# B&R Automation Studio project RSD
Automation Studio 4.3.3.196

## Configuration RSD_Default

CPU X20CP1382, AutomationRuntime I4.33, Build 4.1.2, Vc V4.33.0

### Task classes (Cpu.sw)
```
Cyclic#1 (cycle 2000 us, tolerance 2000 us):
  RSI <- RSI.prg
  Camera <- Camera.prg
Cyclic#2 (cycle 10000 us, tolerance 10000 us):
  Servo <- Servo.prg
  MES_Comm <- MES_Comm.prg
Cyclic#3 (cycle 20000 us, tolerance 20000 us):
  Camera_A <- Camera_A.prg
Cyclic#4:
  Feeder <- Feeder.prg
  Conveyor <- Conveyor.prg
Binaries: udbdef, TCData, ashwac, arconfig, asfw, ashwd, iomap, User, Role, sysconf
Libraries: AsHttp, runtime, AsTCP, AsUDP, standard, MTBasics, brsystem, MTTypes, sys_lib, astime, asieccon
```

### Hardware
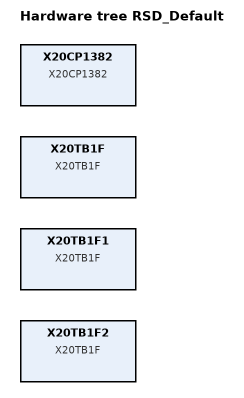
```
X20CP1382 : X20CP1382 v1.3.2.0  [X1 -> X1.SL; X2 -> X2.SL; X3 -> X3.SL]
  Module X1 (Type=X1, Virtual=true, Version=1.3.2.0)
    Connection (Connector=SS1, TargetModule=X20TB1F, TargetConnector=SS)
    Connection (Connector=SL, TargetModule=X20CP1382, TargetConnector=X1)
  Module X2 (Type=X2, Virtual=true, Version=1.3.2.0)
    Connection (Connector=SS1, TargetModule=X20TB1F1, TargetConnector=SS)
    Connection (Connector=SL, TargetModule=X20CP1382, TargetConnector=X2)
  Module X3 (Type=X3, Virtual=true, Version=1.3.2.0)
    Connection (Connector=SS1, TargetModule=X20TB1F2, TargetConnector=SS)
    Connection (Connector=SL, TargetModule=X20CP1382, TargetConnector=X3)
    X3Channel09Source = PWMout
  Connector IF2:
    ActivateDevice = 1
    Mode = Manual
    InternetAddress = 192.168.1.80
    SubnetMask = 255.255.255.0
    InaNodeNumber = 0
  ConfigurationID = RSD_RSD_Default
  SystemTick = 1000
  TaskClassIdleTime = 5000
  CyclicTaskClassCount = 4
  Cyclic1Duration = 2000
  Cyclic1Tolerance = 2000
  Cyclic1Stack = 16384
  Cyclic2Duration = 10000
  Cyclic2Tolerance = 10000
  Cyclic3Duration = 20000
  Cyclic3Tolerance = 20000
X20TB1F : X20TB1F v1.0.0.0
X20TB1F1 : X20TB1F v1.0.0.0
X20TB1F2 : X20TB1F v1.0.0.0
```

### IoMap.iom - X20CP1382/IoMap.iom
```iecst
VAR_CONFIG
	::Camera_A:Camera_trigger AT %QX."X3".DigitalOutput01;
	::Conveyor:Conveyor_out AT %QX."X3".DigitalOutput02;
	::Enable_in AT %IX."X2".DigitalInput01;
	::Sensor_in AT %IX."X2".DigitalInput02;
	::Servo:Period AT %QW."X3".PWMPeriod09;
	::Servo:Pulse AT %QW."X3".PWMOutput09;
	::Feeder:Output_signal AT %QX."X3".DigitalOutput03;
	::Feeder:Enable_feeder AT %IX."X2".DigitalInput09;
END_VAR
```

## Logical view

Binary libraries used (declarations not repeated): operator, runtime, astime, AsIecCon, AsHttp, AsTCP, AsUDP, standard, MTBasics 2.21.0, brsystem, MTTypes 1.03.4, sys_lib, asstring

### Global.var - Global variables
```iecst
VAR
	Camera_bad : BOOL := FALSE;
	Enable_in : BOOL;
	Sensor_in : BOOL;
	Camera_good : BOOL := FALSE;
	Tilt : BOOL := FALSE;
	Data_send : STRING[200] := '';
	Data_recv_vector : ARRAY[0..9] OF STRING[4];
	data_received : BOOL := FALSE;
	New_data : BOOL := FALSE;
	Data_recv_index : USINT := 0;
	Current_part_id : UDINT;
	Part_selected : BOOL := FALSE;
	Data_length : USINT;
	Should_recv : BOOL := FALSE;
	Current_part_post : BOOL := FALSE;
	Robot_index : STRING[2];
	Ready : STRING[1];
	Activate_override : BOOL := TRUE;
	Buffer_use : STRING[1] := '0';
	Activate : BOOL := FALSE;
END_VAR
```

### Global2.typ
```iecst
TYPE
	Variables : 	STRUCT
		isGoodCounter : USINT;
		isBadCounter : USINT;
		position : UDINT;
		sliske : UDINT;
		buffer_bad : ARRAY[0..4]OF UDINT;
		buffer_good : ARRAY[0..10]OF UDINT;
	END_STRUCT;
END_TYPE
```


### Program Logical/Camera_A (IEC)

#### Variables.var
```iecst
VAR
	Delay : MTBasicsTimeDelay;
	Camera_trigger : BOOL := TRUE;
END_VAR
```

#### Main.st
```iecst
PROGRAM _INIT
	(* Insert code here *)
	Delay.Enable := TRUE;
	Delay.DelayTime := 0.227; // 1 at 10hz, 0.4 at 20hz

END_PROGRAM

PROGRAM _CYCLIC
	(* Insert code here *)

	IF Enable_in = TRUE THEN
		Delay.In := BOOL_TO_REAL(Sensor_in);
		Delay();
		Camera_trigger := REAL_TO_BOOL(Delay.Out);
	ELSE
		Camera_trigger := FALSE;
	END_IF

END_PROGRAM

PROGRAM _EXIT
	(* Insert code here *)

END_PROGRAM
```

### Program Logical/Conveyor (IEC)

#### Variables.var
```iecst
VAR
	Conveyor_out : BOOL := FALSE;
END_VAR
```

#### Cyclic.st
```iecst
PROGRAM _CYCLIC
	(* Insert code here *)
	Conveyor_out := Enable_in;

END_PROGRAM
```

#### Init.st
```iecst
PROGRAM _INIT
	(* Insert code here *)

END_PROGRAM
```

### Program Logical/MES_Comm (IEC)

#### Client.st - Cyclic code
```iecst
(********************************************************************
 * COPYRIGHT -- Bernecker + Rainer
 ********************************************************************
 * Program: Client
 * File: Client.st
 * Author: Bernecker + Rainer
 * Created: February 21, 2008
 ********************************************************************
 * Implementation of program Client
 ********************************************************************)
PROGRAM _INIT

END_PROGRAM
PROGRAM _CYCLIC

	CASE Client.sStep OF

		 3: (* IDLE state - waits here until there is something to send *)
			IF New_data <> FALSE THEN
				Client.sStep:=20;
			END_IF;

		 0: (* Open Ethernet Interface *)
			Client.TcpOpen_0.enable := 1;
			Client.TcpOpen_0.pIfAddr := 0;  (* Which Interface to open *)
			Client.TcpOpen_0.port := 13001;  (* Port on client side to use *)
			Client.TcpOpen_0.options :=  0;
			Client.TcpOpen_0;  (* Call the Function *)

			IF Client.TcpOpen_0.status = 0 THEN  (* TcpOpen successfull *)
				Client.sStep := 5;
			ELSIF Client.TcpOpen_0.status = ERR_FUB_BUSY THEN  (* TcpOpen not finished -> redo *)
			  (* Busy *)
			ELSE  (* Goto Error Step *)
				Client.sStep := 100;
			END_IF

		 5:
		 	Client.linger_opt.lLinger := 0; (* linger Time = 0 *)
			Client.linger_opt.lOnOff := 1; (* linger Option ON *)

		 	Client.TcpIoctl_0.enable := 1;
			Client.TcpIoctl_0.ident := Client.TcpOpen_0.ident; (* Connection Ident from AsTP.TCP_Open *)
			Client.TcpIoctl_0.ioctl := tcpSO_LINGER_SET; (* Set Linger Options *)
			Client.TcpIoctl_0.pData := ADR(Client.linger_opt);
			Client.TcpIoctl_0.datalen := SIZEOF(Client.linger_opt);
   			Client.TcpIoctl_0;

			IF Client.TcpIoctl_0.status = 0 THEN  (* TcpIoctl successfull *)
				Client.sStep := 10;
			ELSIF Client.TcpIoctl_0.status = ERR_FUB_BUSY THEN  (* TcpIoctl not finished -> redo *)
			  (* Busy *)
			ELSE  (* Goto Error Step *)
				Client.sStep := 100;
			END_IF

		10: (* Connect to the other Station *)
			Client.TcpClient_0.enable := 1;
			Client.TcpClient_0.ident := Client.TcpOpen_0.ident;  (* Connection Ident from AsTCP.TCP_Open *)
			Client.TcpClient_0.portserv := 4567;  (* Port on server side to use *)
			Client.TcpClient_0.pServer := ADR('192.168.1.23');  (* Server Address *)
			Client.TcpClient_0;  (* Call the Function*)

			IF Client.TcpClient_0.status = 0 THEN  (* Open ok -> Send Data *)
				Client.sStep := 3;
			ELSIF Client.TcpClient_0.status = ERR_FUB_BUSY THEN  (* TcpClient not finished -> redo *)
			  (* Busy *)
			ELSIF Client.TcpClient_0.status = tcpERR_INVALID THEN  (* Port error -> Close actual connection, and reopen a new one *)
				Client.sStep := 40;
			ELSE  (* Goto Error Step *)
				Client.sStep := 100;
			END_IF

		20: (* Send Data to the Server *)
			Client.TcpSend_0.enable := 1;
			Client.TcpSend_0.ident := Client.TcpOpen_0.ident;  (* Connection Ident from AsTCP.TCP_Open *)
			Client.TcpSend_0.pData := ADR(Data_send);  (* Which data to send *)
			Client.TcpSend_0.datalen := Data_length; //SIZEOF(Data_send);  (* Lenght of data to send *)
			Client.TcpSend_0.flags := 0;
			Client.TcpSend_0;  (* Call the Function*)
			Data_recv_index := 0;
			FOR counter:=0 TO 9 BY 1 DO
				Data_recv_vector[counter] := '';
			END_FOR

			IF Client.TcpSend_0.status = 0 THEN  (* Data was sent sucessfully -> receive data *)
				New_data:=FALSE;
				IF Should_recv THEN
					Client.sStep := 30;
				ELSE
					Client.sStep := 3;
				END_IF

			ELSIF Client.TcpSend_0.status = ERR_FUB_BUSY THEN  (* TcpSend not finished -> redo *)
			  (* Busy *)
			ELSIF (Client.TcpSend_0.status = tcpERR_SENTLEN) OR (Client.TcpSend_0.status = tcpERR_NOT_CONNECTED) THEN (* Connection Lost *)
				Client.sStep := 40;
			ELSE  (* Goto Error Step *)
				Client.sStep := 100;
			END_IF

	    30: (* Receive Data from the Server *)
			Client.TcpRecv_0.enable := 1;
			Client.TcpRecv_0.ident := Client.TcpOpen_0.ident;  (* Connection Ident from AsTCP.TCP_Open *)
			Client.TcpRecv_0.pData	:= ADR(Data_recv_vector[Data_recv_index]);  (* Where to store the incoming data *)
			Client.TcpRecv_0.datamax := SIZEOF(Data_recv_vector[Data_recv_index]);  (* Lenght of data buffer *)
			Client.TcpRecv_0.flags := 0;
			Client.TcpRecv_0;  (* Call the Function*)

			IF Client.TcpRecv_0.status = 0 THEN  (* Data was received sucessfully -> Send next packet *)
				Client.sStep := 30;
				Client.recv_timeout := 0;

				//Data_recv_vector[Data_recv_index] := Data_recv;
				Data_recv_index := Data_recv_index +1;
			ELSIF Client.TcpRecv_0.status = tcpERR_NO_DATA THEN  (* No data received - wait *)
				Client.recv_timeout := Client.recv_timeout + 1;
				IF Client.recv_timeout > 10 THEN
					Client.sStep := 3;
					Client.recv_timeout := 0;
					data_received := TRUE;
				END_IF

				(* No Data received *)
			ELSIF Client.TcpRecv_0.status = ERR_FUB_BUSY THEN  (* TcpRecv not finished -> redo *)
				(* Busy *)
			ELSIF Client.TcpRecv_0.status = tcpERR_NOT_CONNECTED THEN (* Connection Lost *)
				Client.sStep := 40;
			ELSE  (* Goto Error Step *)
				Client.sStep := 100;
			END_IF

		40: (* Close connection *)
			Client.TcpClose_0.enable := 1;
			Client.TcpClose_0.ident := Client.TcpOpen_0.ident;  (* Connection Ident from AsTCP.TCP_Open *)
			Client.TcpClose_0.how := 0;
			Client.TcpClose_0;  (* Call the Function*)

			IF Client.TcpClose_0.status = 0 THEN  (* Close sucessfull -> Reopen the interface *)
				Client.sStep := 3;
			ELSIF Client.TcpClose_0.status = ERR_FUB_BUSY THEN  (* TcpClose not finished -> redo *)
			  (* Busy *)
			ELSE  (* Goto Error Step *)
				Client.sStep := 100;
			END_IF

	   100: (* Here some error Handling has to be implemented *)

	END_CASE

END_PROGRAM
```

#### Client.var - Data for Client Task
```iecst
(********************************************************************
 * COPYRIGHT -- Bernecker + Rainer
 ********************************************************************
 * Package: LibAsTCP
 * File: LibAsTCP.var
 * Author: Bernecker + Rainer
 * Created: February 21, 2008
 ********************************************************************
 * Variables of package LibAsTCP
 ********************************************************************)
VAR
	Client : Client_typ := (0); (*Data for Client Task*)
	State_send : USINT := 0;
	counter : USINT;
END_VAR
```

#### Variables.var - not listed in the package file held
```iecst
VAR
	Client : httpClient;
	Enable : BOOL := TRUE;
	Send : BOOL := FALSE;
	IP : STRING[80] := '192.168.1.23';
	URI : STRING[80] := '/plc.test';
	RESPONSE : STRING[4096];
	REQUESTLENGTH : UDINT := 0;
	REQUESTDATA : STRING[80];
	RESPONSELENGTH : UDINT := 4096;
END_VAR
```

#### Cyclic.st - not listed in the package file held
```iecst
PROGRAM _CYCLIC
	(* Insert code here *)
	Client.enable := Enable;

	Client.send := Send;

	Client();

END_PROGRAM
```

#### Init.st - not listed in the package file held
```iecst
PROGRAM _INIT
	(* Insert code here *)
	Client.hostPort := 80;
	Client.method := httpMETHOD_GET;
	Client.option := httpOPTION_HTTP_11;
	Client.pHost := ADR(IP);
	Client.pUri := ADR(URI);
	Client.pRequestData := ADR(REQUESTDATA);
	Client.requestDataLen := REQUESTLENGTH;
	Client.pResponseData := ADR(RESPONSE);
	Client.responseDataSize := RESPONSELENGTH;

END_PROGRAM
```

### Program Logical/MES_machine (IEC)

#### Main.st - Init, cyclic, exit code
```iecst
PROGRAM _INIT
	(* Insert code here *)

END_PROGRAM

PROGRAM _CYCLIC
	(* Insert code here *)

	CASE MES_step OF

		0:		// ST-Start
			Part_selected := FALSE;
			data_received := FALSE;

		5:		// ST-Idle
			IF Order_selected = FALSE THEN
				MES_step := 20;

			ELSIF Part_selected = FALSE AND Sensor_in THEN
				MES_step := 10;

			ELSIF Current_part_post = FALSE AND (Camera_good OR Camera_bad) THEN
				MES_step := 15;

			ELSIF Part_status_posted THEN
				IF Camera_good AND Order_good > 0 THEN
					MES_step := 30;
				ELSIF Camera_bad AND Order_bad > 0 THEN
					MES_step := 30;
				ELSIF Camera_good AND buffer_free(ADR(variables), TRUE) THEN
					MES_step := 40;
				ELSIF Camera_bad AND buffer_free(ADR(variables), FALSE) THEN
					MES_step := 40;
				ELSE
					MES_step := 43;

				END_IF

				Part_status_posted := FALSE;
			END_IF

		10:		// ST-Get part
			IF New_data = FALSE THEN
				Data_send := 'GET PART 1$n';
				Data_length := 11;
				New_data := TRUE;
				MES_step := 11;
				Should_recv := TRUE;
				Activate_override := TRUE;
			END_IF

		11:
			IF data_received = TRUE THEN
				data_received := FALSE;
				memcpy(ADR(Current_part_id), ADR(Data_recv_vector[0]),4);
				Part_selected := TRUE;
				Current_part_post := FALSE;
				MES_step := 5;
			END_IF

		15:		// ST-Post Part
			IF New_data = FALSE THEN
				Data_send := 'POST PARTSTATUS$n';
				Number := 1000;
				WHILE Number > Current_part_id AND Number <> 0 DO
					Data_send:=CONCAT(Data_send, '0');
					Number := Number/10;
				END_WHILE;

				IF Current_part_id <> 0 THEN
					String_tmp := UDINT_TO_STRING(Current_part_id);
					Data_send:=CONCAT(Data_send, String_tmp);
				END_IF

				IF Camera_good THEN
					Data_send:=CONCAT(Data_send, ' 1$n');
				ELSIF Camera_bad THEN
					Data_send:=CONCAT(Data_send, ' 0$n');
				END_IF

				Data_length := 23;
				Should_recv := FALSE;
				New_data := TRUE;
				Part_selected := FALSE;
				Current_part_post := TRUE;
				MES_step := 5;
				Part_status_posted := TRUE;
			END_IF

		20:		// ST-Get Order
			IF New_data = FALSE THEN
				Data_send := 'GET ORDER 1$n';
				Data_length := 12;
				Current_order_ids := '';
				New_data := TRUE;
				MES_step := 21;
				Should_recv := TRUE;
			END_IF

		21:
			IF data_received = TRUE THEN
				data_received := FALSE;
				memcpy(ADR(Current_order_id), ADR(Data_recv_vector[0]),4);
				IF Current_order_id > 10000 THEN
					MES_step := 45;
				ELSE
					Order_good := 0;
					Order_bad := 0;
					memcpy(ADR(Current_order_parts), ADR(Data_recv_vector[1]),4);
					FOR Order_index:=0 TO Current_order_parts-1 BY 1 DO
						memcpy(ADR(Parts_vector[Order_index]), ADR(Data_recv_vector[Order_index+2]),4);
						IF Parts_vector[Order_index] = 1 THEN
							Order_good := Order_good +1;
						ELSIF Parts_vector[Order_index] = 0 THEN
							Order_bad := Order_bad +1;
						END_IF

					END_FOR

					Order_selected := TRUE;
						MES_step := 5;

				END_IF

			END_IF

		25:		// ST-Post Order
			IF New_data = FALSE THEN
				Data_send := 'POST ORDERSTATUS$n';
				Number := 1000;
				WHILE Number > Current_order_id AND Number <> 0 DO
					Data_send:=CONCAT(Data_send, '0');
					Number := Number/10;
				END_WHILE;

				IF Current_order_id <> 0 THEN
					String_tmp := UDINT_TO_STRING(Current_order_id);
					Data_send:=CONCAT(Data_send, String_tmp);
				END_IF

				Data_length := 21;
				Data_send := CONCAT(Data_send, Current_order_ids);
				Current_order_ids := CONCAT(Current_order_ids, 'p');
				Pos_find := FIND(Current_order_ids, 'p');
				Data_length := Data_length + INT_TO_USINT(Pos_find);

				Data_send := CONCAT(Data_send, '$n');
				Should_recv := FALSE;
				New_data := TRUE;
				Order_selected := FALSE;
				MES_step := 5;
			END_IF

		30:		// ST - Put box
			Buffer_use := '0';
			Robot_index := '0';
			String_tmp := UDINT_TO_STRING(Current_part_id);
			Current_order_ids := CONCAT(Current_order_ids, String_tmp);
			Current_order_ids := CONCAT(Current_order_ids, ' ');
			IF Camera_good THEN
				Order_good := Order_good - 1;
			ELSIF Camera_bad THEN
				Order_bad := Order_bad -1;
			END_IF;
			MES_step := 31;

		31:
			IF Ready = '0' THEN
				MES_step := 32;
			END_IF;

		32:
			IF Ready = '1' THEN
				IF Order_good = 0 AND Order_bad = 0 THEN
					Tilt := TRUE;
					MES_step := 25;
				ELSIF Order_good > 0 AND in_buffer(ADR(variables),TRUE) THEN
					MES_step := 35;
				ELSIF Order_bad > 0 AND in_buffer(ADR(variables), FALSE) THEN
					MES_step := 35;
				ELSE
					MES_step := 5;
				END_IF

			END_IF;

		35:		// ST- Tak Buf
			Buffer_use := '0';
			IF Order_good > 0 AND in_buffer(ADR(variables), TRUE) THEN
				Robot_index := UDINT_TO_STRING(fetch_brick_decimal(ADR(variables), TRUE));
				Buffer_part_id := get_partid(ADR(variables), TRUE, variables.isGoodCounter);
				Order_good := Order_good - 1;
			ELSIF Order_bad > 0 AND in_buffer(ADR(variables), FALSE) THEN
				Robot_index := UDINT_TO_STRING(fetch_brick_decimal(ADR(variables), FALSE));
				Buffer_part_id := get_partid(ADR(variables), FALSE, variables.isBadCounter);
				Order_bad := Order_bad - 1;
			END_IF

			Activate := TRUE;

			String_tmp := UDINT_TO_STRING(Buffer_part_id);
			Current_order_ids := CONCAT(Current_order_ids, String_tmp);
			Current_order_ids := CONCAT(Current_order_ids, ' ');
			MES_step := 36;

		36:
			IF Ready = '0' THEN
				MES_step := 37;
			END_IF

		37:
			IF Ready = '1' THEN
				IF Order_good = 0 AND Order_bad = 0 THEN
					Tilt := TRUE;
					MES_step := 25;
				ELSE
					MES_step := 5;
				END_IF
			END_IF

		40:		// ST- put buf

			IF Camera_good AND buffer_free(ADR(variables), TRUE) THEN
				Buffer_use := '1';
				Robot_index := UDINT_TO_STRING(save_brick_decimal(ADR(variables), TRUE, Current_part_id));
			ELSIF Camera_bad AND buffer_free(ADR(variables), FALSE) THEN
				Buffer_use := '1';
				Robot_index := UDINT_TO_STRING(save_brick_decimal(ADR(variables), FALSE, Current_part_id));
			END_IF
			MES_step := 41;

		41:
			IF Ready = '0' THEN
				MES_step := 42;
			END_IF;

		42:
			IF Ready = '1' THEN
				MES_step := 5;
			END_IF

		43: // BUF full
			Activate_override := FALSE;

			IF New_data = FALSE THEN
				Data_send := 'POST PARTSTATUS$n';
				Number := 1000;
				WHILE Number > Current_part_id AND Number <> 0 DO
					Data_send:=CONCAT(Data_send, '0');
					Number := Number/10;
				END_WHILE;

				IF Current_part_id <> 0 THEN
					String_tmp := UDINT_TO_STRING(Current_part_id);
					Data_send:=CONCAT(Data_send, String_tmp);
				END_IF

				Data_send:= CONCAT(Data_send, ' Buffer full$n');

				Data_length := 33;
				Should_recv := FALSE;
				New_data := TRUE;
				MES_step := 5;
			END_IF

		45:		// ST- Finished
			Activate_override := FALSE;

	END_CASE

END_PROGRAM

PROGRAM _EXIT
	(* Insert code here *)

END_PROGRAM
```

#### Variables2.var - Local variables
```iecst
VAR
	MES_step : USINT := 0;
	Number : UDINT;
	Pos_find : INT;
	String_tmp : STRING[200];
	Current_order_id : UDINT;
	Order_selected : BOOL := FALSE;
	Current_order_parts : UDINT;
	Order_index : UDINT;
	Parts_vector : ARRAY[0..4] OF UDINT;
	Order_good : UDINT;
	Order_bad : UDINT;
	Part_status_posted : BOOL := FALSE;
	Current_order_ids : STRING[200];
	Part_moved : BOOL := FALSE;
	Buffer_part_id : UDINT;
END_VAR
```

#### buffer_free.st
```iecst
(* TODO: Add your comment here *)
FUNCTION buffer_free
	IF type THEN
		IF var.isGoodCounter < 10 THEN
			buffer_free:= TRUE;
		ELSE
			buffer_free:=FALSE;
		END_IF;
	END_IF;

	IF type = FALSE THEN
		IF var.isBadCounter < 5 THEN
			buffer_free:= TRUE;
		ELSE
			buffer_free:=FALSE;
		END_IF;
	END_IF;
END_FUNCTION
```

#### fetch_brick.st
```iecst
FUNCTION fetch_brick
	IF type THEN
		IF var.isGoodCounter <> 0 THEN
			fetch_brick:=var.isGoodCounter;
			var.isGoodCounter:=var.isGoodCounter-1;
		ELSE
			fetch_brick:=-1; // Empty
		END_IF;
	ELSE
		IF var.isBadCounter <> 0 THEN
			fetch_brick:=var.isBadCounter;
			var.isBadCounter:=var.isBadCounter-1;
		ELSE
			fetch_brick:=-1; // Empty
		END_IF;
	END_IF;
END_FUNCTION
```

#### fetch_brick_decimal.st
```iecst
(* TODO: Add your comment here *)
FUNCTION fetch_brick_decimal
	var.position := fetch_brick(ADR(var), type);

	IF var.position = -1 THEN
		fetch_brick_decimal := -1;
		RETURN;
	END_IF;

	IF type = FALSE THEN
		var.sliske:=2;
	ELSE
		IF var.position > 5 THEN
			var.sliske:=3;
		ELSE
			var.sliske:=1;
		END_IF;
	END_IF;

	IF var.position > 5 THEN
		fetch_brick_decimal := SHL(var.sliske,3) + var.position -5 -1;
	ELSE
		fetch_brick_decimal := SHL(var.sliske,3) + var.position -1;
	END_IF

END_FUNCTION
```

#### get_partid.st
```iecst
(* TODO: Add your comment here *)
FUNCTION get_partid
	IF type THEN
		get_partid:=var.buffer_good[pos];
	END_IF;

	IF type = FALSE THEN
		get_partid:=var.buffer_bad[pos];
	END_IF;
END_FUNCTION
```

#### in_buffer.st
```iecst
(* TODO: Add your comment here *)
FUNCTION in_buffer
	IF type THEN
		IF var.isGoodCounter > 0 THEN
			in_buffer:=TRUE;
		ELSE
			in_buffer:=FALSE;
		END_IF;
	END_IF;

	IF type = FALSE THEN
		IF var.isBadCounter > 0 THEN
			in_buffer:=TRUE;
		ELSE
			in_buffer:=FALSE;
		END_IF;
	END_IF;
END_FUNCTION
```

#### LocalFunctions.fun
```iecst
FUNCTION get_partid : UDINT
	VAR_INPUT
		var : REFERENCE TO Variables;
		type : BOOL;
		pos : UDINT;
	END_VAR
END_FUNCTION

FUNCTION fetch_brick : UDINT (*TODO: Add your comment here*) (*$GROUP=User,$CAT=User,$GROUPICON=User.png,$CATICON=User.png*)
	VAR_INPUT
		var : REFERENCE TO Variables;
		type : BOOL;
	END_VAR
END_FUNCTION

FUNCTION save_brick : UDINT (*TODO: Add your comment here*) (*$GROUP=User,$CAT=User,$GROUPICON=User.png,$CATICON=User.png*)
	VAR_INPUT
		var : REFERENCE TO Variables;
		type : BOOL;
		partid : UDINT;
	END_VAR
END_FUNCTION

FUNCTION fetch_brick_decimal : UDINT (*TODO: Add your comment here*) (*$GROUP=User,$CAT=User,$GROUPICON=User.png,$CATICON=User.png*)
	VAR_INPUT
		var : REFERENCE TO Variables;
		type : BOOL;
	END_VAR
END_FUNCTION

FUNCTION save_brick_decimal : UDINT (*TODO: Add your comment here*) (*$GROUP=User,$CAT=User,$GROUPICON=User.png,$CATICON=User.png*)
	VAR_INPUT
		var : REFERENCE TO Variables;
		type : BOOL;
		partid : UDINT;
	END_VAR
END_FUNCTION

FUNCTION buffer_free : BOOL
	VAR_INPUT
		var : REFERENCE TO Variables;
		type : BOOL;
	END_VAR
END_FUNCTION

FUNCTION in_buffer : BOOL
	VAR_INPUT
		var : REFERENCE TO Variables;
		type : BOOL;
	END_VAR
END_FUNCTION
```

#### save_brick.st
```iecst
FUNCTION save_brick
	IF type THEN
		IF var.isGoodCounter < 10 THEN
			var.buffer_good[var.isGoodCounter] := partid;
			var.isGoodCounter:=var.isGoodCounter+1;
			save_brick:=var.isGoodCounter;
		ELSE
			save_brick:=-1; // Full
		END_IF;
	ELSE
		IF var.isBadCounter < 4 THEN
			var.buffer_bad[var.isBadCounter]:= partid;
			var.isBadCounter:=var.isBadCounter+1;
			save_brick:=var.isBadCounter;
		ELSE
			save_brick:=-1; // Full
		END_IF;
	END_IF;
END_FUNCTION
```

#### save_brick_decimal.st
```iecst
(* TODO: Add your comment here *)
FUNCTION save_brick_decimal
	var.position := save_brick(ADR(var), type, partid);

	IF var.position = -1 THEN
		save_brick_decimal := -1;
		RETURN;
	END_IF;

	IF type = FALSE THEN
		var.sliske:=2;
	ELSE
		IF var.position > 5 THEN
			var.sliske:=3;
		ELSE
			var.sliske:=1;
		END_IF;
	END_IF;

	IF var.position > 5 THEN
		save_brick_decimal := SHL(var.sliske,3) + var.position -5 -1;
	ELSE
		save_brick_decimal := SHL(var.sliske,3) + var.position -1;
	END_IF

END_FUNCTION
```

#### Variables.var - Local variables
```iecst
VAR
	test : UDINT := 0;
	variables : Variables;
	isgood : BOOL;
END_VAR
```

### Program Logical/Camera (IEC)

#### LibAsTCP1_ST.typ - Global Datatype
```iecst
(********************************************************************
 * COPYRIGHT -- Bernecker + Rainer
 ********************************************************************
 * Package: LibAsTCP
 * File: LibAsTCP.typ
 * Author: Bernecker + Rainer
 * Created: February 21, 2008
 ********************************************************************
 * Data types of package LibAsTCP
 ********************************************************************)

TYPE
	LibAsTCP1_ST_typ : 	STRUCT  (*Datatyp for global Variables*)
		receive_data : STRING[80]; (*Data which has been received*)
		Bad : UDINT := 0;
		Good : UDINT := 0;
	END_STRUCT;
END_TYPE
```

#### Client.st - Cyclic code
```iecst
(********************************************************************
 * COPYRIGHT -- Bernecker + Rainer
 ********************************************************************
 * Program: Client
 * File: Client.st
 * Author: Bernecker + Rainer
 * Created: February 21, 2008
 ********************************************************************
 * Implementation of program Client
 ********************************************************************)

PROGRAM _CYCLIC

	CASE Client.sStep OF

		 0: (* Open Ethernet Interface *)
			Client.TcpOpen_0.enable := 1;
			Client.TcpOpen_0.pIfAddr := 0;  (* Which Interface to open *)
			Client.TcpOpen_0.port := 12001;  (* Port on client side to use *)
			Client.TcpOpen_0.options := 0;
			Client.TcpOpen_0;  (* Call the Function *)

			IF Client.TcpOpen_0.status = 0 THEN  (* TcpOpen successfull *)
				Client.sStep := 5;
			ELSIF Client.TcpOpen_0.status = ERR_FUB_BUSY THEN  (* TcpOpen not finished -> redo *)
			  (* Busy *)
			ELSE  (* Goto Error Step *)
				Client.sStep := 100;
			END_IF

		 5:
		 	Client.linger_opt.lLinger := 0; (* linger Time = 0 *)
			Client.linger_opt.lOnOff := 1; (* linger Option ON *)

		 	Client.TcpIoctl_0.enable := 1;
			Client.TcpIoctl_0.ident := Client.TcpOpen_0.ident; (* Connection Ident from AsTP.TCP_Open *)
			Client.TcpIoctl_0.ioctl := tcpSO_LINGER_SET; (* Set Linger Options *)
			Client.TcpIoctl_0.pData := ADR(Client.linger_opt);
			Client.TcpIoctl_0.datalen := SIZEOF(Client.linger_opt);
   			Client.TcpIoctl_0;

			IF Client.TcpIoctl_0.status = 0 THEN  (* TcpIoctl successfull *)
				Client.sStep := 10;
			ELSIF Client.TcpIoctl_0.status = ERR_FUB_BUSY THEN  (* TcpIoctl not finished -> redo *)
			  (* Busy *)
			ELSE  (* Goto Error Step *)
				Client.sStep := 100;
			END_IF

		10: (* Connect to the other Station *)
			Client.TcpClient_0.enable := 1;
			Client.TcpClient_0.ident := Client.TcpOpen_0.ident;  (* Connection Ident from AsTCP.TCP_Open *)
			Client.TcpClient_0.portserv := 9876;  (* Port on server side to use *)
			Client.TcpClient_0.pServer := ADR('192.168.1.10');  (* Server Address *)
			Client.TcpClient_0;  (* Call the Function*)

			IF Client.TcpClient_0.status = 0 THEN  (* Open ok -> Send Data *)
				Client.sStep := 30;
			ELSIF Client.TcpClient_0.status = ERR_FUB_BUSY THEN  (* TcpClient not finished -> redo *)
			  (* Busy *)
			ELSIF Client.TcpClient_0.status = tcpERR_INVALID THEN  (* Port error -> Close actual connection, and reopen a new one *)
				Client.sStep := 40;
			ELSE  (* Goto Error Step *)
				Client.sStep := 100;
			END_IF

	    30: (* Receive Data from the Server *)
			Client.TcpRecv_0.enable := 1;
			Client.TcpRecv_0.ident := Client.TcpOpen_0.ident;  (* Connection Ident from AsTCP.TCP_Open *)
			Client.TcpRecv_0.pData	:= ADR(LibAsTCP1_ST.receive_data);  (* Where to store the incoming data *)
			Client.TcpRecv_0.datamax := SIZEOF(LibAsTCP1_ST.receive_data);  (* Lenght of data buffer *)
			Client.TcpRecv_0.flags := 0;
			Client.TcpRecv_0;  (* Call the Function*)

			IF Client.TcpRecv_0.status = 0 THEN  (* Data was received sucessfully -> Send next packet *)
				Client.sStep := 30;
				IF LibAsTCP1_ST.receive_data = '     0.0000$r' THEN
					LibAsTCP1_ST.Good := LibAsTCP1_ST.Good +1;
					Camera_good := TRUE;
				ELSIF LibAsTCP1_ST.receive_data = '    -1.0000$r' THEN
					Camera_bad := TRUE;
					LibAsTCP1_ST.Bad := LibAsTCP1_ST.Bad + 1;
				END_IF;

			ELSIF Client.TcpRecv_0.status = tcpERR_NO_DATA THEN  (* No data received - wait *)
				(* No Data received *)
			ELSIF Client.TcpRecv_0.status = ERR_FUB_BUSY THEN  (* TcpRecv not finished -> redo *)
				(* Busy *)
			ELSIF Client.TcpRecv_0.status = tcpERR_NOT_CONNECTED THEN (* Connection Lost *)
				Client.sStep := 40;
			ELSE  (* Goto Error Step *)
				Client.sStep := 100;
			END_IF

		40: (* Close connection *)
			Client.TcpClose_0.enable := 1;
			Client.TcpClose_0.ident := Client.TcpOpen_0.ident;  (* Connection Ident from AsTCP.TCP_Open *)
			Client.TcpClose_0.how := 0;
			Client.TcpClose_0;  (* Call the Function*)

			IF Client.TcpClose_0.status = 0 THEN  (* Close sucessfull -> Reopen the interface *)
				Client.sStep := 0;
			ELSIF Client.TcpClose_0.status = ERR_FUB_BUSY THEN  (* TcpClose not finished -> redo *)
			  (* Busy *)
			ELSE  (* Goto Error Step *)
				Client.sStep := 100;
			END_IF

		100: (* Here some error Handling has to be implemented *)
			Client.sStep := 40;

	END_CASE

END_PROGRAM
```

### Program Logical/RSI (IEC)

#### Server.typ - UDP Server Variables
```iecst
(********************************************************************
 * COPYRIGHT -- Bernecker + Rainer
 ********************************************************************
 * Program: Server
 * File: Server.typ
 * Author: Bernecker + Rainer
 * Created: June 02, 2008
 ********************************************************************
 * Local data types of program Server
 ********************************************************************)

TYPE
	Server_typ : 	STRUCT  (*UDP Server Variables*)
		sStep : UINT; (*UDP Server Step Variable*)
		client_address : STRING[20]; (*Address of the client connection to the Server*)
		UdpOpen_0 : UdpOpen; (*AsUDP.UdpOpen FUB*)
		UdpConnect_0 : UdpConnect; (*AsUDP.UdpConnect FUB*)
		UdpSend_0 : UdpSend; (*AsUDP.UdpSend FUB*)
		UdpRecv_0 : UdpRecv; (*AsUDP.UdpRecv FUB*)
		UdpDisconnect_0 : UdpDisconnect; (*AsUDP.UdpDisconnect FUB*)
		UdpClose_0 : UdpClose; (*AsUDP.UdpClose FUB*)
		data_buffer : STRING[200]; (*Data buffer ( receive and send )*)
	END_STRUCT;
END_TYPE
```

#### Server.var - Data for Server Task
```iecst
(********************************************************************
 * COPYRIGHT -- Bernecker + Rainer
 ********************************************************************
 * Program: Server
 * File: Server.var
 * Author: Bernecker + Rainer
 * Created: June 02, 2008
 ********************************************************************
 * Local variables of program Server
 ********************************************************************)
VAR
	Server : Server_typ := (0); (*Data for Server Task*)
	startPos : INT;
	TOC : STRING[50];
	endPos : INT;
	Output : STRING[500];
	Delay : MTBasicsTimeDelay;
	Old_delay : REAL := 0.0;
	Counting : USINT := 0;
	Old_Ready : STRING[1] := '1';
	Buffer_test : STRING[5] := '0';
	Buffer_bad : ARRAY[0..3] OF STRING[2];
	Buffer_good : ARRAY[0..9] OF STRING[2];
	index_good : USINT := 0;
	Good_brick : BOOL := FALSE;
	index_bad : USINT := 0;
END_VAR
```

#### Server.st - Cyclic code
```iecst
(********************************************************************
 * COPYRIGHT -- Bernecker + Rainer
 ********************************************************************
 * Program: Server
 * File: Server.st
 * Author: Bernecker + Rainer
 * Created: June 02, 2008
 ********************************************************************
 * Implementation of program Server
 ********************************************************************)

PROGRAM _CYCLIC

	IF Enable_in = TRUE THEN
		IF Camera_good OR Camera_bad THEN
			Delay.In := 1.0;
		ELSE
			Delay.In := 0.0;
		END_IF

		Delay();

		IF Delay.Out = 1.0 AND Old_delay = 0.0 THEN
			Old_delay := 1.0;
			Activate := TRUE;
			Camera_good := FALSE;
			Camera_bad := FALSE;
		ELSIF Delay.Out = 0.0 THEN
			Old_delay := 0.0;
		END_IF

	ELSE
		Activate := FALSE;
	END_IF

	IF Ready = '0' THEN
		Activate := FALSE;
	END_IF

	CASE Server.sStep OF

		0:	(* Open UDP Port *)
			Server.UdpOpen_0.enable := 1;
			Server.UdpOpen_0.pIfAddr := 0;	(* Listen on all TCP/IP Interfaces*)
			Server.UdpOpen_0.port := 49000;	(* Port to listen*)
			Server.UdpOpen_0.options := 0;
			Server.UdpOpen_0;	(* Call the Function*)

			IF Server.UdpOpen_0.status = 0 THEN  (* UdpOpen successful*)
				Server.sStep := 1;
			ELSIF Server.UdpOpen_0.status = ERR_FUB_BUSY THEN  (* UdpOpen not finished -> redo *)
			  (* Busy *)
			ELSE  (* Goto Error Step *)
				Server.sStep := 10;
			END_IF

		1:	(* Wait for Data *)
			Server.UdpRecv_0.enable := 1;
			Server.UdpRecv_0.ident := Server.UdpOpen_0.ident;	(* Client Ident from AsUDP.UDP_Open *)
			Server.UdpRecv_0.pData := ADR(Server.data_buffer);	(* Where to store the incoming data *)
			Server.UdpRecv_0.datamax := SIZEOF(Server.data_buffer);	(* Lenght of data buffer *)
			Server.UdpRecv_0.flags := 0;
			Server.UdpRecv_0.pIpAddr := ADR(Server.client_address);	(* IP Address of the Client *)
			Server.UdpRecv_0;	(* Call the Function*)

			IF Server.UdpRecv_0.status = 0 THEN  (* Data received *)
				Server.sStep := 2;
				Ready:=MID(Server.data_buffer,1,25);

			ELSIF Server.UdpRecv_0.status = udpERR_NO_DATA THEN  (* No data received - wait *)
				(* No Data received *)
			ELSIF Server.UdpRecv_0.status = ERR_FUB_BUSY THEN  (* UdpRecv not finished -> redo *)
				(* Busy *)
			ELSE  (* Goto Error Step *)
				Server.sStep := 10;
			END_IF

		2:	(* Send Data back to Client *)
			startPos:=FIND(Server.data_buffer,'<IPOC>');
				endPos:=FIND(Server.data_buffer, '</Rob>');

				TOC:=MID(Server.data_buffer,endPos-startPos,startPos);

			Output:='<Sen Type="ImFree"><Activate>';

			IF Enable_in = TRUE AND Ready = '1' AND Activate = TRUE AND Activate_override THEN

				//IF Activate = TRUE THEN
				Output:=CONCAT(Output, '1');
			ELSE
				Output:=CONCAT(Output, '0');
			END_IF

			Output:=CONCAT(Output,'</Activate>');
			Output:=CONCAT(Output,'<Buf>');
			Output:=CONCAT(Output,Buffer_use);
			Output:=CONCAT(Output,'</Buf>');
			Output:=CONCAT(Output,'<Index>');
			Output:=CONCAT(Output, Robot_index);

			//IF Good_brick AND Activate THEN
			//	Output:=CONCAT(Output,Buffer_good[index_good]);
			//	index_good := index_good +1;
			//	Activate:=FALSE;
			//ELSIF Good_brick = FALSE AND Activate THEN
			//	Output:=CONCAT(Output,Buffer_bad[index_bad]);
			//	index_bad := index_bad +1;
			//	Activate:=FALSE;
			//ELSE
			//	Output:=CONCAT(Output,'0');
			//END_IF

			//test
			//IF Activate THEN
			//	Output:=CONCAT(Output, Buffer_test);
			//	Activate := FALSE;
			//END_IF;

			Output:=CONCAT(Output,'</Index>');
			Output:=CONCAT(Output, TOC);
			Output:=CONCAT(Output,'</Sen>');

			// 100 -> robot ready -> to PLC
			// 101 -> Activate -> to Robot
			// 102 -> Buf -> to Robot
			// 113-128 -> Index (word 16 bit) -> to Robot

			Server.UdpSend_0.enable := 1;
			Server.UdpSend_0.ident := Server.UdpOpen_0.ident;	(* Client Ident from AsUDP.UDP_Open *)
			Server.UdpSend_0.pHost := ADR(Server.client_address);	(* IP Address of the Client *)
			Server.UdpSend_0.port := Server.UdpRecv_0.port;		(* Port number of the Client *)
			Server.UdpSend_0.pData := ADR(Output);	(* Which data to send *)
			Server.UdpSend_0.datalen := SIZEOF(Output);	(* Lenght of data to send *)
			Server.UdpSend_0.flags := 0;
			Server.UdpSend_0;	(* Call the Function*)

			IF Server.UdpSend_0.status = 0 THEN  (* Data sent *)
				Server.sStep := 1;
			ELSIF Server.UdpSend_0.status = ERR_FUB_BUSY THEN  (* UdpSend not finished -> redo *)
			  (* Busy *)
			ELSE  (* Goto Error Step *)
				Server.sStep := 10;
			END_IF

		10:  (* Here some error Handling has to be implemented *)

	END_CASE

END_PROGRAM
```

#### Init.st
```iecst
PROGRAM _INIT
	(* Insert code here *)

	Delay.Enable := TRUE;
	Delay.DelayTime := 0.2; // 2.25 at 10hz, 1.125 at 20hz

	Buffer_good[0] := '8';
	Buffer_good[1] := '9';
	Buffer_good[2] := '10';
	Buffer_good[3] := '11';
	Buffer_good[4] := '12';
	Buffer_good[5] := '24';
	Buffer_good[6] := '25';
	Buffer_good[7] := '26';
	Buffer_good[8] := '27';
	Buffer_good[9] := '28';

	Buffer_bad[0] := '16';
	Buffer_bad[1] := '17';
	Buffer_bad[2] := '18';
	Buffer_bad[3] := '19';

END_PROGRAM
```

### Program Logical/Servo (IEC)

#### Variables.var
```iecst
VAR
	Period : {REDUND_UNREPLICABLE} UINT := 20000;
END_VAR
VAR CONSTANT
	Duty_cycle_pos2 : INT := 37;
	Duty_cycle_pos1 : INT := 130;
END_VAR
VAR
	Pulse : INT;
	Delay : MTBasicsTimeDelay;
END_VAR
```

#### Cyclic.st
```iecst
PROGRAM _CYCLIC
	(* Insert code here *)
	IF Tilt = TRUE THEN
		Pulse := Duty_cycle_pos1;
		// Delay.In :=
		Delay.In := 1.0;
	END_IF
	Delay();
	IF Delay.Out = 1.0 THEN
		Pulse := Duty_cycle_pos2;
		Delay.In := 0.0;
		Tilt := FALSE;
	END_IF

	(* call function block *)

END_PROGRAM
```

#### Init.st
```iecst
PROGRAM _INIT

	Delay.Enable := TRUE;
	Delay.DelayTime := 1;
END_PROGRAM
```

### Program Logical/Feeder (IEC)

#### Variables.var
```iecst
VAR
	Counter : USINT := 0;
	Output_signal : BOOL := FALSE;
	Enable_feeder : BOOL := FALSE;
END_VAR
```

#### Main.st
```iecst
PROGRAM _INIT
	(* Insert code here *)

END_PROGRAM

PROGRAM _CYCLIC
	(* Insert code here *)

	IF Enable_feeder AND Enable_in THEN
		IF Counter = 60 THEN
			Output_signal := NOT Output_signal;
			Counter := 0;
		END_IF

		Counter := Counter +1;
	ELSE
		Output_signal := FALSE;
	END_IF;

END_PROGRAM

PROGRAM _EXIT
	(* Insert code here *)

END_PROGRAM
```

### Program Logical/Im_alive

#### Variables.var
```iecst
VAR
	alive_led : BOOL := TRUE;
END_VAR
```

#### Main.st
```iecst
PROGRAM _INIT
	(* Insert code here *)

END_PROGRAM

PROGRAM _CYCLIC
	(* Insert code here *)

	alive_led := Sensor_in;
END_PROGRAM

PROGRAM _EXIT
	(* Insert code here *)

END_PROGRAM
```

Listed in the project but not available here: Logical/Global.typ, Logical/MES_Comm/Client.typ, Logical/MES_machine/Types2.typ, Logical/MES_machine/Types.typ, Logical/Camera/LibAsTCP1_ST.var, Logical/Camera/Client.typ, Logical/Camera/Client.var
